// TwinCAT 3 PLC project Untitled1
// ProgramVersion: 3.1.4023.0
// libraries:
//   Tc2_Standard, * (Beckhoff Automation GmbH)
//   Tc2_System, * (Beckhoff Automation GmbH)
//   Tc3_Database, * (Beckhoff Automation GmbH)
//   Tc3_Module, * (Beckhoff Automation GmbH)
// project tree:
//   DUTs/ st_InsertData.TcDUT, st_ReturnedData.TcDUT
//   / PlcTask.TcTTO
//   POUs/ fb_CSVRead.TcPOU, fb_CreateTable.TcPOU, fb_CSVWrite.TcPOU, fb_datareturn.TcPOU, fb_InsertRecord.TcPOU, MAIN.TcPOU

CONFIGURATION Untitled1
    RESOURCE PLC ON TwinCAT3
        TASK PlcTask(INTERVAL := T#10ms, PRIORITY := 20);
        PROGRAM MAIN WITH PlcTask : MAIN;
    END_RESOURCE
END_CONFIGURATION

// ---- DUTs/st_InsertData.TcDUT
TYPE st_InsertData :
STRUCT
	Datum:STRING(100);
	temp_set:STRING(10);
	temp_act:STRING(10);
	hum_set:STRING(10);
	hum_act:STRING(10);
END_STRUCT
END_TYPE

// ---- DUTs/st_ReturnedData.TcDUT
TYPE st_ReturnedData :
STRUCT
//	Datum:STRING(255);
	//temp_set:LINT;
	//temp_act:LINT;
	//hum_set:LINT;
	//hum_act:LINT;
		Datum:DATE_AND_TIME;
	temp_set:DINT;
	temp_act:DINT;
	hum_set:DINT;
	hum_act:DINT;
END_STRUCT
END_TYPE

// ---- POUs/MAIN.TcPOU
PROGRAM MAIN
VAR
	nstep:INT:=20;
	connection:FB_sqlcommandevt(snetid:='', tTimeout:=T#5S);
	
	Datareturn:fb_datareturn;
	createtable:fb_createtable;
	insertRecord:fb_insertrecord;
	WriteCSV: fb_CSVWrite;
	ReadCSV:fb_CSVRead;
	
	st_insertdata:ST_insertdata;
	bDataReturn:BOOL:=FALSE;
	bCreateTable:BOOL:=FALSE;
	bInsert:BOOL:=FALSE;
	
	dbid:UINT:=3;
	table:STRING:='$'1_kamra$'';
	start:STRING:='$'2020-07-01 15:00:01$'';
	end:STRING:='$'2020-08-30 15:00:01$'';
	
END_VAR

CASE nstep OF 
	
	20:
		IF bdatareturn THEN
			datareturn.ClearArray();
			nstep:=30;
			bdatareturn:=FALSE;
		END_IF
		IF bCreateTable THEN
			nstep:=40;
			bcreatetable:=FALSE;
		END_IF
		IF bInsert THEN
			nstep:=50;
			bInsert:=FALSE;
		END_IF
		
		
		
	30:	// datareturn
		
		datareturn(dbid:=dbid,
					table:=table,
					start:=start,
					end:=end,
					bexecute:=TRUE);
		IF datareturn.Error THEN
			nstep:=99;
		ELSE
		IF datareturn.bReady THEN
			
			nstep:=20;
			datareturn.Reset();
		END_IF
		END_IF
		
	40:	//create table
		createtable(table:=table,
					bExecute:=TRUE,
					DBID:=dbid);
		IF createtable.bError THEN
			nstep:=99;
		ELSE	
		IF createtable.bReady THEN
			createtable.Reset();	
			nstep:=20;
		END_IF
		END_IF
	50: // insert data
		//st_insertData.Datum:='$'2020-01-01 12:00:20$'';//DT#2020-07-28-15:00:01 ;
		////st_insertdata.hum_act:='1';
		//st_insertdata.hum_set:='2';
		//st_insertdata.temp_act:='3';
		//st_insertdata.temp_set:='4';
		insertrecord(insertdata:=st_insertdata,
					table:=table,
					DBID:=dbid,
					bExecute:=TRUE);
		IF insertrecord.bError THEN
			nstep:=99;
		ELSE
		IF insertrecord.bReady THEN
			nstep:=20;
			insertrecord.Reset();
		END_IF
		END_IF

	60: // write csv
		st_insertData.Datum:='2020-01-01 12:00:20';//DT#2020-07-28-15:00:01 ;
		st_insertdata.hum_act:='1';
		st_insertdata.hum_set:='2';
		st_insertdata.temp_act:='3';
		st_insertdata.temp_set:='4';
		WriteCSV(dbid:=4,
				table:='1_kamra',
				bExecute:=TRUE);
		IF WriteCSV.bError THEN
			nstep:=99;
		ELSE
		IF  WriteCSV.bReady THEN
			nstep:=20;
			WriteCSV.reset();
		END_IF
		END_IF		
	
	70:	//ReadCSV
		ReadCSV(dbid:=4,
				table:='1_kamra',
				bExecute:=TRUE);
		IF ReadCSV.bError THEN
			nstep:=99;
		ELSE
		IF  ReadCSV.bReady THEN
			nstep:=20;
			ReadCSV.reset();
		END_IF
		END_IF		
	99:// error
		;	
			
END_CASE

END_PROGRAM

// ---- POUs/fb_datareturn.TcPOU
FUNCTION_BLOCK fb_datareturn
VAR_INPUT
	dbid:UINT;
	table:STRING(50);
	start:STRING(100);
	end:STRING(100);
	bExecute:BOOL;
	
	
END_VAR
VAR_OUTPUT
	ReadStruct: ARRAY [0..1700] OF ST_ReturnedData;
	bReady:BOOL:=FALSE;
	Error:BOOL:=FALSE;
END_VAR
VAR
	sCmd:STRING(255):='';
	nstep:int:=10;
	SQLresult: FB_SQLResultEvt(sNetID:='', tTimeout:=T#5S);
	SQLcommand: FB_SQLCommandEvt(sNetid:='',tTimeout:=T#5S);
	Connectdb: FB_sqldatabaseevt(SNetID:='', tTimeout:=T#5S);
	//bExecute:BOOL:=FALSE;
	connected:BOOL:=FALSE;
	
END_VAR

	
		
IF bExecute THEN
	CASE nstep OF
	10:
				sCmd:=CONCAT('SELECT * FROM ',table);
				sCmd:=concat(sCmd, ' WHERE Dátum BETWEEN ');
				sCmd:=concat(sCmd , start);
				sCmd:=Concat(sCmd , ' AND ');
				sCmd:=concat(sCmd , end);
				sCmd:=concat(sCmd,';');
				nstep:=20;
	20:		IF connectDB.Connect(dbid) THEN
				IF connectdb.bError THEN
					Error:=TRUE;
				ELSE
					connected:=TRUE;
					nstep:=25;
				END_IF
			END_IF
		//	IF connected AND NOT connectDB.bBusy THEN 
			//	IF connectDB.CreateCmd(pSQLCommand:= ADR(SQLcommand)) THEN
			//		nstep:=30;
			//	END_IF
		//	END_IF	
		
			
	25:		IF connected THEN
				IF connectDB.CreateCmd(pSQLCommand:= ADR(SQLcommand)) THEN
					nstep:=30;
				END_IF
			END_IF						
	30:
			IF SQLcommand.ExecuteDataReturn(pSQLCmd:=ADR(sCmd),
										cbSQLCmd:=SIZEOF(sCmd),
										pSQLDBResult:=ADR(SQLResult))
			THEN
			IF sqlcommand.bError THEN
				Error:=TRUE;
			ELSE
				nstep:=40;
			END_IF
			END_IF
	40:	IF SQLResult.Read(nStartindex:= 1,
						  nRecordCount:=1001,
						  pData:=ADR(ReadStruct),
						  cbData:=SIZEOF(ReadStruct),
							TRUE, TRUE)
		THEN
		IF sqlresult.bError THEN
			Error:=TRUE;
		ELSE
			nstep:=45;
		END_IF
		END_IF	
	
	50:
		IF connectDB.Disconnect() THEN
			IF connectdb.bError THEN
				Error:=TRUE;
			ELSE
				connected:=FALSE;
				bReady:=TRUE;
				bExecute:=FALSE;	
		END_IF
		END_IF	
END_CASE
END_IF

METHOD ClearArray : BOOL
VAR_INPUT
END_VAR
memset(adr(readstruct),0,sizeof(readstruct));
END_METHOD

METHOD Reset : BOOL
VAR_INPUT
END_VAR
bReady:=FALSE;
nstep:=10;
END_METHOD

END_FUNCTION_BLOCK

// ---- POUs/fb_CreateTable.TcPOU
FUNCTION_BLOCK fb_CreateTable
VAR_INPUT
	table:STRING(50);
	bExecute:BOOL;
	DBID:UINT;
	
END_VAR
VAR_OUTPUT
	bError:BOOL:=FALSE;
	bReady:BOOL:=FALSE;
END_VAR
VAR
	sCmd:STRING(255);
	nstep:INT:=10;
	SQLcommand: FB_SQLCommandEvt(sNetid:='',tTimeout:=T#5S);
	Connectdb: FB_sqldatabaseevt(SNetID:='', tTimeout:=T#5S);
	connected:BOOL:=FALSE;
END_VAR

IF bExecute THEN
CASE nstep OF
	10:
		IF connectDB.Connect(DBID) THEN
			
			IF connectdb.bError THEN
				bError:=TRUE;
			ELSE
				connected:=TRUE;	
			END_IF
		END_IF
		IF connected and NOT connectDB.bBusy THEN 
			IF connectDB.CreateCmd(pSQLCommand:= ADR(SQLcommand)) THEN
				nstep:=20;
			END_IF
		END_IF
	20:	
	
		sCmd:=concat('CREATE TABLE ', table);
		sCmd:=concat(sCmd,'(Dátum DATETIME ,
  						temp_set INTEGER ,
  						temp_act INTEGER ,
  						hum_set INTEGER ,
 						 hum_act INTEGER );');
		nstep:=30;
		
	30:
		IF SQLcommand.Execute(pSQLCmd:=ADR(sCmd),
							cbSQLCmd:=SIZEOF(sCmd))
		THEN
			IF sqlcommand.bError THEN
				berror:=TRUE;
			ELSE
			IF NOT SQLcommand.bBusy THEN
				nstep:=40;
			
			END_IF
			END_IF
		END_IF
	40:	
		IF connectDB.Disconnect() THEN
			IF connectdb.bError THEN
				bError:=TRUE;
			ELSE
				connected:=FALSE;
			bReady:=TRUE;
			bExecute:=FALSE;	
		END_IF
		END_IF	
			
END_CASE
END_IF

METHOD Reset : BOOL
VAR_INPUT
END_VAR
bReady:=FALSE;
nstep:=10;
END_METHOD

END_FUNCTION_BLOCK

// ---- POUs/fb_InsertRecord.TcPOU
FUNCTION_BLOCK fb_InsertRecord
VAR_INPUT
	InsertData:ST_InsertData;
	table:STRING(50);
	DBID:UINT;
	bExecute:BOOL;
	
END_VAR
VAR_OUTPUT
	bError:BOOL:=FALSE;
	bReady:BOOL:=FALSE;
	
END_VAR
VAR
	nstep:INT:=10;
	sCmd:STRING(255);
	SQLcommand: FB_SQLCommandEvt(sNetid:='',tTimeout:=T#5S);
	Connectdb: FB_sqldatabaseevt(SNetID:='', tTimeout:=T#5S);
	connected:BOOL:=FALSE;
	
END_VAR

IF bExecute THEN
CASE nstep OF 
	10:
			sCmd:=concat('insert into ',table);
			sCmd:=concat(sCmd,  ' (Dátum , temp_set, temp_act, hum_set, hum_act ) values ('); //{Datum},{temp_set},{temp_act},{hum_set}, {hum_act})');
			sCmd:=concat(sCmd,insertdata.Datum);
			sCmd:=concat(sCmd,', ');
			sCmd:=concat(sCmd,insertdata.temp_set);
			sCmd:=concat(sCmd,', ');
			sCmd:=concat(sCmd,insertdata.temp_act);
			sCmd:=concat(sCmd,', ');
			sCmd:=concat(sCmd, insertdata.hum_set);
			sCmd:=concat(sCmd,', ');
			sCmd:=concat(sCmd,insertdata.hum_act);
			sCmd:=concat(sCmd,')');
			nstep:=20;
	20:
			IF connectDB.Connect(DBID) THEN
				IF connectdb.bError THEN
					bError:=TRUE;
				ELSE
					connected:=TRUE;	
				END_IF
			END_IF
			IF connected AND NOT connectDB.bBusy THEN 
				IF connectDB.CreateCmd(pSQLCommand:= ADR(SQLcommand)) THEN
					nstep:=30;
				END_IF
			END_IF		
	30:
		IF SQLcommand.Execute(pSQLCmd:=ADR(sCmd),
							cbSQLCmd:=SIZEOF(sCmd))
			THEN
			IF sqlcommand.bError THEN
				Berror:=TRUE;
			ELSE
			IF NOT SQLcommand.bBusy THEN
				nstep:=40;
			END_IF
			END_IF
		END_IF
	40:	
		IF connectDB.Disconnect() THEN
			IF connectdb.bError THEN
				bError:=TRUE;
			ELSE
				connected:=FALSE;
				bReady:=TRUE;
				bExecute:=FALSE;	
		END_IF
		END_IF		
		
END_CASE
END_IF

METHOD Reset : BOOL
VAR_INPUT
END_VAR
bReady:=FALSE;
nstep:=10;
END_METHOD

END_FUNCTION_BLOCK

// ---- POUs/fb_CSVWrite.TcPOU
FUNCTION_BLOCK fb_CSVWrite
VAR_INPUT
	bExecute:BOOL;
	dbid:UINT;
	table:STRING(100);
END_VAR
VAR_OUTPUT
	bError:BOOL:=FALSE;
	bReady:BOOL:=FALSE;
END_VAR
VAR
	PLCDBWrite:fb_PLCDBWrite(snetid:='', tTimeout:=T#15S);
	Columnnames: ARRAY [0..4] OF STRING(50):=['Dátum', 'temp_set', 'temp_act', 'hum_set', 'hum_act'];
	InsertData:ST_InsertData;
	
	
	
END_VAR

IF bExecute THEN
	IF PLCDBWrite.WriteStruct(hDBID:=dbid,
							stablename:=table,
							pRecord:=ADR(InsertData),
							cbRecord:=SIZEOF(InsertData),
							pColumnNames:=ADR(columnNames),
							cbColumnNames:=SIZEOF(columnNames))
	THEN
	IF plcdbwrite.bError THEN
		bError:=TRUE;
		
	ELSE 
	IF NOT plcdbwrite.bBusy THEN
		bExecute:=FALSE;
		bReady:=TRUE;
	END_IF
	END_IF
END_IF	
	
							
END_IF

METHOD Reset : BOOL
VAR_INPUT
END_VAR
BReady:=false;
END_METHOD

END_FUNCTION_BLOCK

// ---- POUs/fb_CSVRead.TcPOU
FUNCTION_BLOCK fb_CSVRead
VAR_INPUT
	bExecute:BOOL;
	dbid:UINT;
	table:STRING(100);
END_VAR
VAR_OUTPUT
	bError:BOOL:=FALSE;
	bReady:BOOL:=FALSE;
END_VAR
VAR
	PLCDBRead:fb_PLCDBRead(sNetid:='', tTimeOut:=T#15S);
	ReadStruct: ARRAY [0..1700] OF ST_ReturnedData;
	Columnnames: ARRAY [0..4] OF STRING(50):=['Dátum', 'temp_set', 'temp_act', 'hum_set', 'hum_act'];
END_VAR

IF bExecute THEN
	IF PLCDBread.ReadStruct(hDBID:=dbid,
							sTableName:=table,
							pColumnNames:=ADR(ColumnNames),
							cbColumnNames:=SIZEOF(ColumnNames),
							sOrderByColumn:='Dátum',
							eOrderType:=E_ordertype.ASC,
							nStartIndex:=0,
							nRecordCount:=1000,
							pData:=ADR(readstruct),
							cbData:=SIZEOF(readstruct))
	THEN
	IF plcdbread.bError THEN
		berror:=TRUE;	
	ELSE
	IF NOT plcdbread.bBusy THEN
		bExecute:=FALSE;
		bReady:=TRUE;
	END_IF	
	END_IF
	END_IF				
END_IF

METHOD ClearArray : BOOL
VAR_INPUT
END_VAR
memset(adr(readstruct),0,sizeof(readstruct));
END_METHOD

METHOD reset : BOOL
VAR_INPUT
END_VAR
bReady:=false;
END_METHOD

END_FUNCTION_BLOCK
